// TIA Portal V16 export
// export: Created 2021-11-12T13:33:14.9788844Z, ExportSetting WithDefaults, DisplayName Totally Integrated Automation Portal, DisplayVersion V16 Update 3, DisplayName TIA Portal Version Control Interface, DisplayVersion V16 Update 2, DisplayName TIA Portal Openness, DisplayVersion V16 Update 3, DisplayName SINAMICS Startdrive Advanced, DisplayVersion V16 Update 5, DisplayName SINAMICS Startdrive G130, G150, S120, S150, SINAMICS MV, S210, DisplayVersion V16 Update 5, DisplayName SINAMICS Startdrive G110M, G120, G120C, G120D, G120P, G115D, DisplayVersion V16 Update 5, DisplayName STEP 7 Professional, DisplayVersion V16 Update 3, DisplayName STEP 7 Safety, DisplayVersion V16, DisplayName WinCC UA Professional, DisplayVersion V16 Update 3
DATA_BLOCK "STATUS_Zone400"   // DB120
{ S7_Optimized_Access := 'TRUE'; DB_Accessible_From_OPC_UA := 'FALSE' }
VERSION : 0.1
// stored: AutoNumber true, DBAccessibleFromOPCUA false, IsOnlyStoredInLoadMemory false, IsRetainMemResEnabled false, IsWriteProtectedInAS false, MemoryReserve 100
   VAR
      Mode : Struct   // Statuses and error of zone 400
         Main : "UDT_Status_main";
         Specific : "UDT_Zone_Status_specific";
         Error : "UDT_Error01";
      END_STRUCT;
      Station410_Mode : Struct   // Statuses and error of station 410
         Main : "UDT_Status_main";
         Specific : "UDT_Zone_Status_specific";
         Error : "UDT_Error01";
      END_STRUCT;
      Station420_Mode : Struct   // Statuses and error of station 420
         Main : "UDT_Status_main";
         Specific : "UDT_Zone_Status_specific";
         Error : "UDT_Error01";
      END_STRUCT;
      Station430_Mode : Struct   // Statuses and error of station 430
         Main : "UDT_Status_main";
         Specific : "UDT_Zone_Status_specific";
         Error : "UDT_Error01";
      END_STRUCT;
      Station440_Mode : Struct   // Statuses and error of station 440
         Main : "UDT_Status_main";
         Specific : "UDT_Zone_Status_specific";
         Error : "UDT_Error01";
      END_STRUCT;
      Station450_Mode : Struct   // Statuses and error of station 450
         Main : "UDT_Status_main";
         Specific : "UDT_Zone_Status_specific";
         Error : "UDT_Error01";
      END_STRUCT;
      Station460_Mode : Struct   // Statuses and error of station 460
         Main : "UDT_Status_main";
         Specific : "UDT_Zone_Status_specific";
         Error : "UDT_Error01";
      END_STRUCT;
      StationTHM1_Mode : Struct   // Statuses and error of station THM1
         Main : "UDT_Status_main";
         Specific : "UDT_Zone_Status_specific";
         Error : "UDT_Error01";
      END_STRUCT;
      StationTHM2_Mode : Struct   // Statuses and error of station THM2
         Main : "UDT_Status_main";
         Specific : "UDT_Zone_Status_specific";
         Error : "UDT_Error01";
      END_STRUCT;
   END_VAR
BEGIN
END_DATA_BLOCK
